(* Logix 5000 project; controller SX_V040001_C001 vendor 1 type 14 code 77 rev 16.23; software revision 16.04; part 10 of 35 *)
(* tags used below, declared in another part *)
   ALL_KINDS : INT[90];
   CMD : INT[36];
   command_value : INT;
   DATAOP : INT[10];
   DRIVE : INT[32];
   DRIVE_INTERVAL : INT[8];
   EMPTYING : INT[18];
   G_DInput : DINT[3];
   G_DOutput : DINT[3];
   loading : INT[19];
   louvre : INT[11];
   METERING : INT[44];
   METERING_PULSE : DINT[14];
   NOTDOS : INT[6];
   PARAMETER : INT[501];
   RECIPE_GENERAL : INT[405];
   RM_CMD : INT[9];
   T_CURRENT_EM_METER : TIMER;
   T_DELTA_EM_METER : TIMER;
   T_RPM_EM_METER : TIMER;
   T_TEMP_EM_METER : TIMER;
   TEMP : INT[14];
(* MainProgram, continued *)

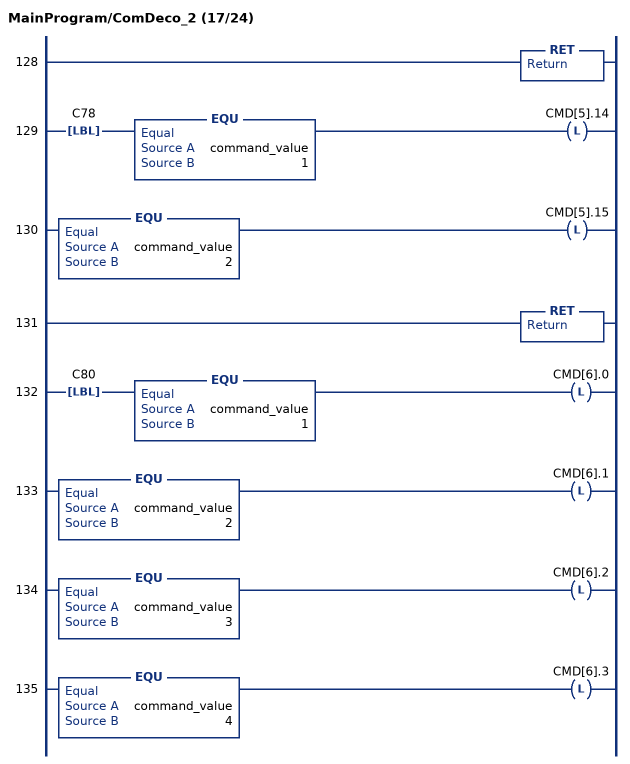
   [picture p205: MainProgram/ComDeco_2 rungs 128-135]
   128: RET();
   129: LBL(C78)EQU(command_value,1)OTL(CMD[5].14);
   130: EQU(command_value,2)OTL(CMD[5].15);
   131: RET();
   132: LBL(C80)EQU(command_value,1)OTL(CMD[6].0);
   133: EQU(command_value,2)OTL(CMD[6].1);
   134: EQU(command_value,3)OTL(CMD[6].2);
   135: EQU(command_value,4)OTL(CMD[6].3);
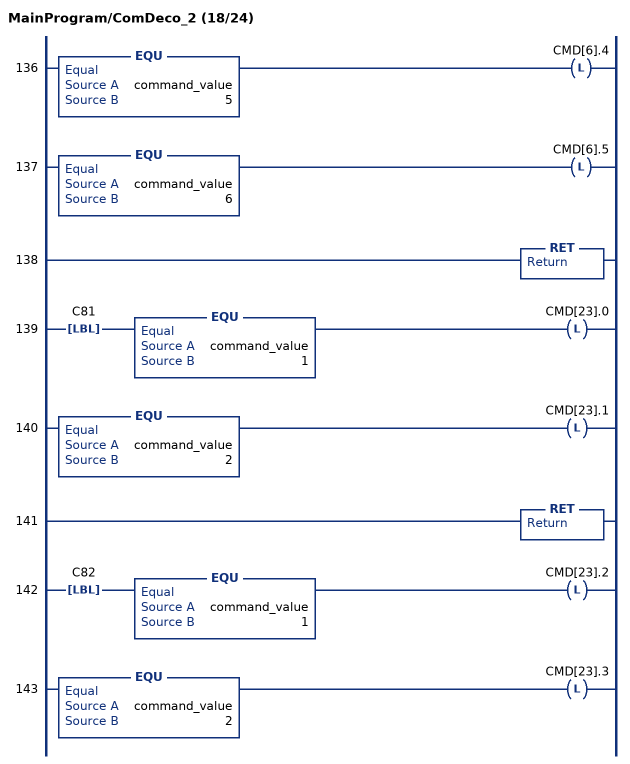
   136: EQU(command_value,5)OTL(CMD[6].4);
   137: EQU(command_value,6)OTL(CMD[6].5);
   138: RET();
   139: LBL(C81)EQU(command_value,1)OTL(CMD[23].0);
   140: EQU(command_value,2)OTL(CMD[23].1);
   141: RET();
   142: LBL(C82)EQU(command_value,1)OTL(CMD[23].2);
   143: EQU(command_value,2)OTL(CMD[23].3);
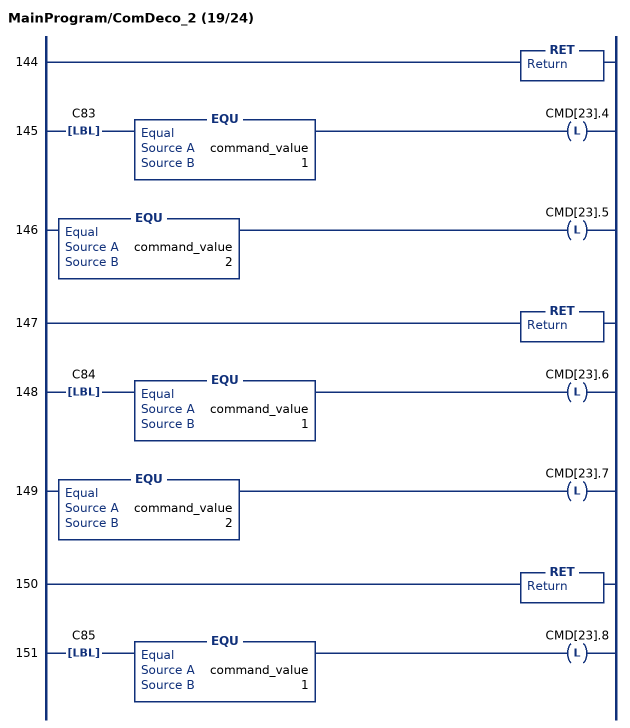
   144: RET();
   145: LBL(C83)EQU(command_value,1)OTL(CMD[23].4);
   146: EQU(command_value,2)OTL(CMD[23].5);
   147: RET();
   148: LBL(C84)EQU(command_value,1)OTL(CMD[23].6);
   149: EQU(command_value,2)OTL(CMD[23].7);
   150: RET();
   151: LBL(C85)EQU(command_value,1)OTL(CMD[23].8);
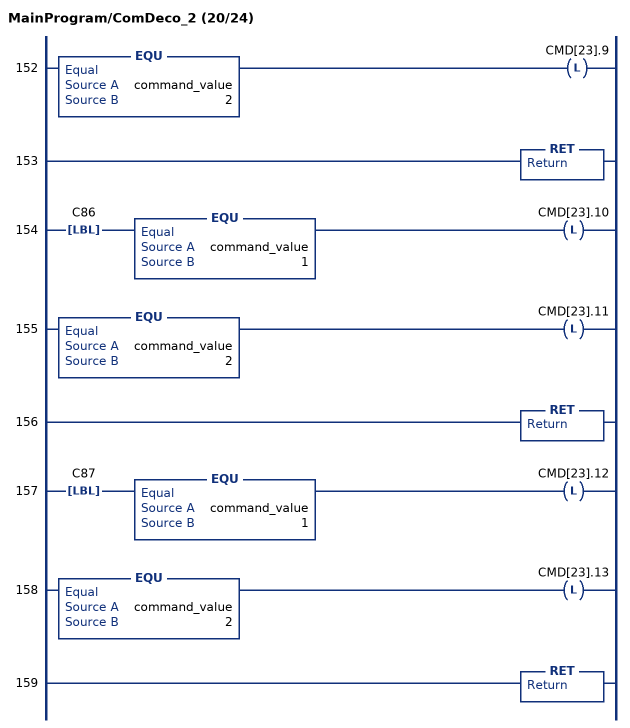
   152: EQU(command_value,2)OTL(CMD[23].9);
   153: RET();
   154: LBL(C86)EQU(command_value,1)OTL(CMD[23].10);
   155: EQU(command_value,2)OTL(CMD[23].11);
   156: RET();
   157: LBL(C87)EQU(command_value,1)OTL(CMD[23].12);
   158: EQU(command_value,2)OTL(CMD[23].13);
   159: RET();
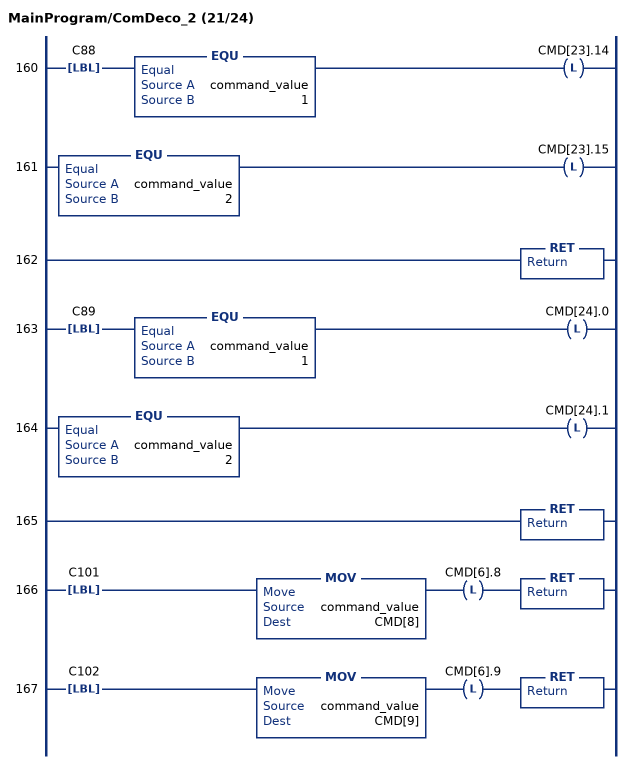
   160: LBL(C88)EQU(command_value,1)OTL(CMD[23].14);
   161: EQU(command_value,2)OTL(CMD[23].15);
   162: RET();
   163: LBL(C89)EQU(command_value,1)OTL(CMD[24].0);
   164: EQU(command_value,2)OTL(CMD[24].1);
   165: RET();
   166: LBL(C101)MOV(command_value,CMD[8])OTL(CMD[6].8)RET();
   167: LBL(C102)MOV(command_value,CMD[9])OTL(CMD[6].9)RET();
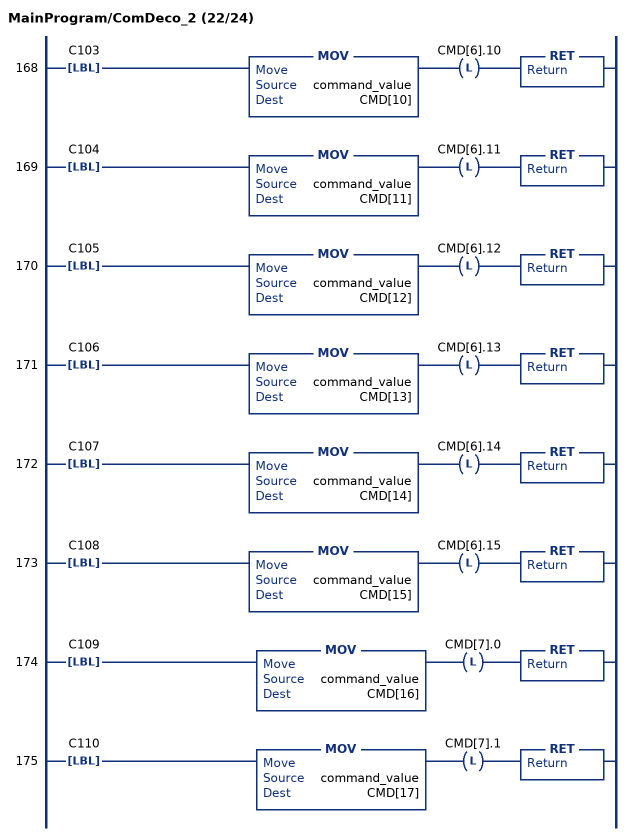
   168: LBL(C103)MOV(command_value,CMD[10])OTL(CMD[6].10)RET();
   169: LBL(C104)MOV(command_value,CMD[11])OTL(CMD[6].11)RET();
   170: LBL(C105)MOV(command_value,CMD[12])OTL(CMD[6].12)RET();
   171: LBL(C106)MOV(command_value,CMD[13])OTL(CMD[6].13)RET();
   172: LBL(C107)MOV(command_value,CMD[14])OTL(CMD[6].14)RET();
   173: LBL(C108)MOV(command_value,CMD[15])OTL(CMD[6].15)RET();
   174: LBL(C109)MOV(command_value,CMD[16])OTL(CMD[7].0)RET();
   175: LBL(C110)MOV(command_value,CMD[17])OTL(CMD[7].1)RET();
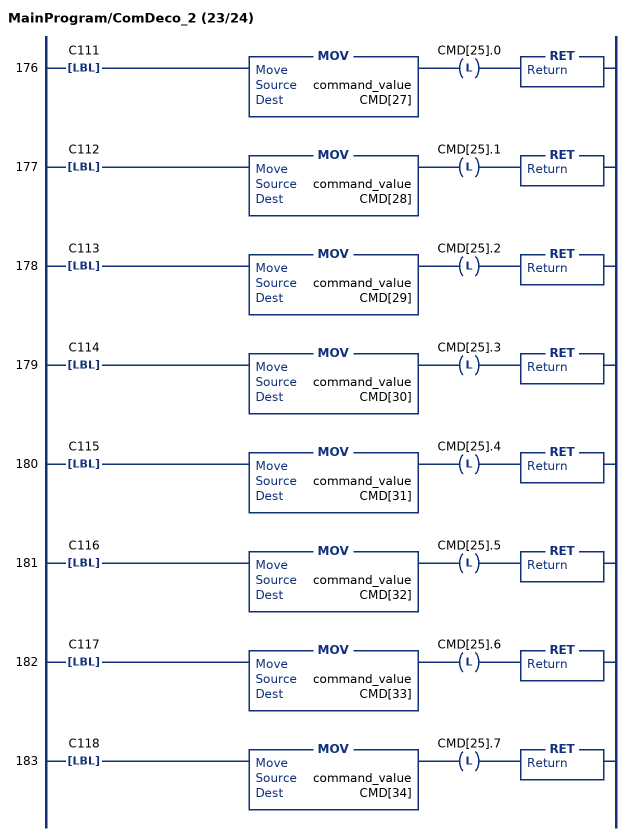
   176: LBL(C111)MOV(command_value,CMD[27])OTL(CMD[25].0)RET();
   177: LBL(C112)MOV(command_value,CMD[28])OTL(CMD[25].1)RET();
   178: LBL(C113)MOV(command_value,CMD[29])OTL(CMD[25].2)RET();
   179: LBL(C114)MOV(command_value,CMD[30])OTL(CMD[25].3)RET();
   180: LBL(C115)MOV(command_value,CMD[31])OTL(CMD[25].4)RET();
   181: LBL(C116)MOV(command_value,CMD[32])OTL(CMD[25].5)RET();
   182: LBL(C117)MOV(command_value,CMD[33])OTL(CMD[25].6)RET();
   183: LBL(C118)MOV(command_value,CMD[34])OTL(CMD[25].7)RET();
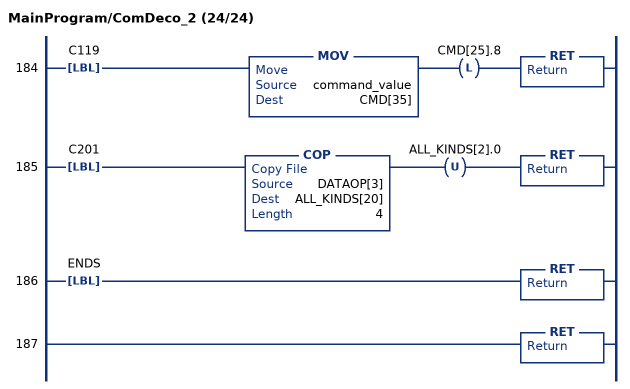
   184: LBL(C119)MOV(command_value,CMD[35])OTL(CMD[25].8)RET();
   185: LBL(C201)COP(DATAOP[3],ALL_KINDS[20],4)OTU(ALL_KINDS[2].0)RET();
   186: LBL(ENDS)RET();
   187: RET();
END_ROUTINE

ROUTINE DeleteData   (* ladder *)
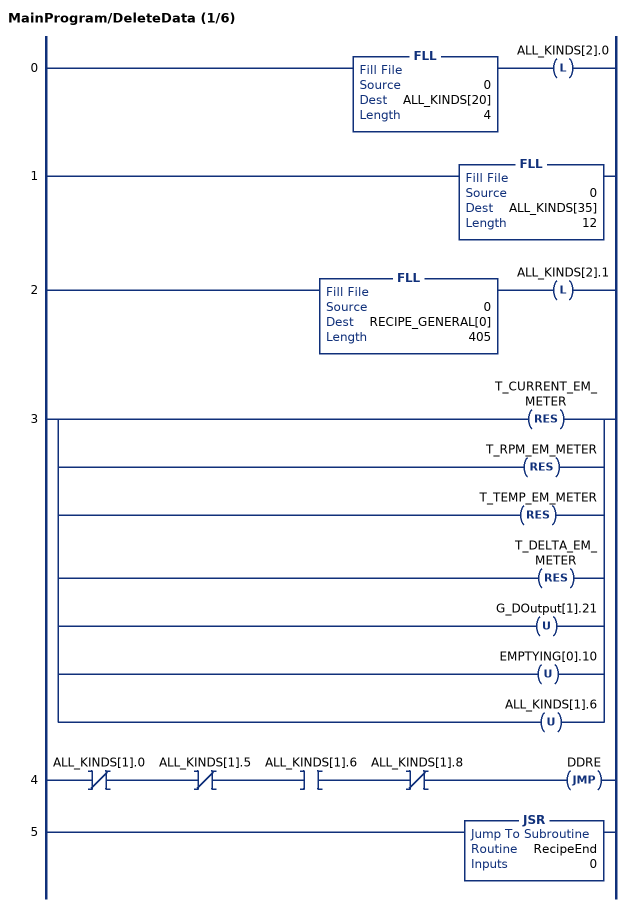
   0: FLL(0,ALL_KINDS[20],4)OTL(ALL_KINDS[2].0);
   1: FLL(0,ALL_KINDS[35],12);
   2: FLL(0,RECIPE_GENERAL[0],405)OTL(ALL_KINDS[2].1);
   3: [RES(T_CURRENT_EM_METER) ,RES(T_RPM_EM_METER) ,RES(T_TEMP_EM_METER) ,RES(T_DELTA_EM_METER) ,OTU(G_DOutput[1].21) ,OTU(EMPTYING[0].10) ,OTU(ALL_KINDS[1].6) ];
   4: XIO(ALL_KINDS[1].0)XIO(ALL_KINDS[1].5)XIC(ALL_KINDS[1].6)XIO(ALL_KINDS[1].8)JMP(DDRE);
   5: JSR(RecipeEnd,0);
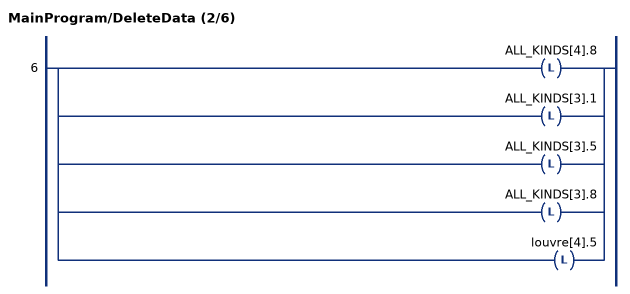
   6: [OTL(ALL_KINDS[4].8) ,OTL(ALL_KINDS[3].1) ,OTL(ALL_KINDS[3].5) ,OTL(ALL_KINDS[3].8) ,OTL(louvre[4].5) ];
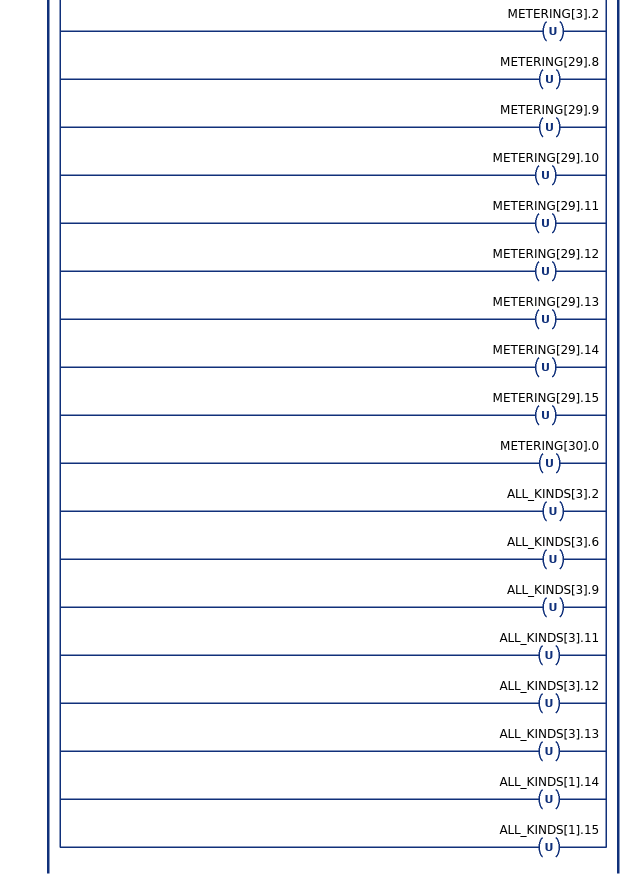
   7: [OTU(ALL_KINDS[4].9) ,OTU(ALL_KINDS[1].3) ,OTU(ALL_KINDS[3].5) ,OTU(ALL_KINDS[1].5) ,OTU(ALL_KINDS[1].7) ,OTU(ALL_KINDS[1].8) ,OTU(ALL_KINDS[1].9) ,OTU(RM_CMD[3].1) ,OTU(ALL_KINDS[1].11) ,OTU(ALL_KINDS[1].12) ,OTU(ALL_KINDS[1].13) ,OTU(ALL_KINDS[2].2) ,OTU(ALL_KINDS[2].4) ,OTU(METERING[2].5) ,OTU(METERING[2].6) ,OTU(EMPTYING[1].9) ,OTU(DRIVE[2].4) ,OTU(DRIVE_INTERVAL[1].0) ,OTU(EMPTYING[0].15) ,OTU(EMPTYING[1].15) ,OTU(TEMP[1].2) ,OTU(loading[1].1) ,OTU(NOTDOS[1].0) ,OTU(NOTDOS[1].7) ,OTU(NOTDOS[1].9) ,OTU(NOTDOS[1].1) ,OTU(NOTDOS[1].8) ,OTU(NOTDOS[1].10) ,OTU(NOTDOS[1].2) ,OTU(NOTDOS[1].3) ,OTU(NOTDOS[1].4) ,OTU(NOTDOS[1].5) ,OTU(NOTDOS[1].6) ,OTU(METERING[1].0) ,OTU(METERING[1].1) ,OTU(METERING[1].2) ,OTU(METERING[1].3) ,OTU(METERING[1].4) ,OTU(METERING[27].0) ,OTU(METERING[27].1) ,OTU(METERING[27].2) ,OTU(METERING[27].3) ,OTU(METERING[27].4) ,OTU(METERING[27].5) ,OTU(METERING[27].6) ,OTU(METERING[27].7) ,OTU(METERING[27].8) ,OTU(METERING[1].10) ,OTU(METERING[1].11) ,OTU(METERING[1].12) ,OTU(METERING[1].13) ,OTU(METERING[1].14) ,OTU(METERING[28].4) ,OTU(METERING[28].5) ,OTU(METERING[28].6) ,OTU(METERING[28].7) ,OTU(METERING[28].8) ,OTU(METERING[28].9) ,OTU(METERING[28].10) ,OTU(METERING[28].11) ,OTU(METERING[28].12) ,OTU(METERING[2].14) ,OTU(METERING[2].15) ,OTU(METERING[3].0) ,OTU(METERING[3].1) ,OTU(METERING[3].2) ,OTU(METERING[29].8) ,OTU(METERING[29].9) ,OTU(METERING[29].10) ,OTU(METERING[29].11) ,OTU(METERING[29].12) ,OTU(METERING[29].13) ,OTU(METERING[29].14) ,OTU(METERING[29].15) ,OTU(METERING[30].0) ,OTU(ALL_KINDS[3].2) ,OTU(ALL_KINDS[3].6) ,OTU(ALL_KINDS[3].9) ,OTU(ALL_KINDS[3].11) ,OTU(ALL_KINDS[3].12) ,OTU(ALL_KINDS[3].13) ,OTU(ALL_KINDS[1].14) ,OTU(ALL_KINDS[1].15) ];
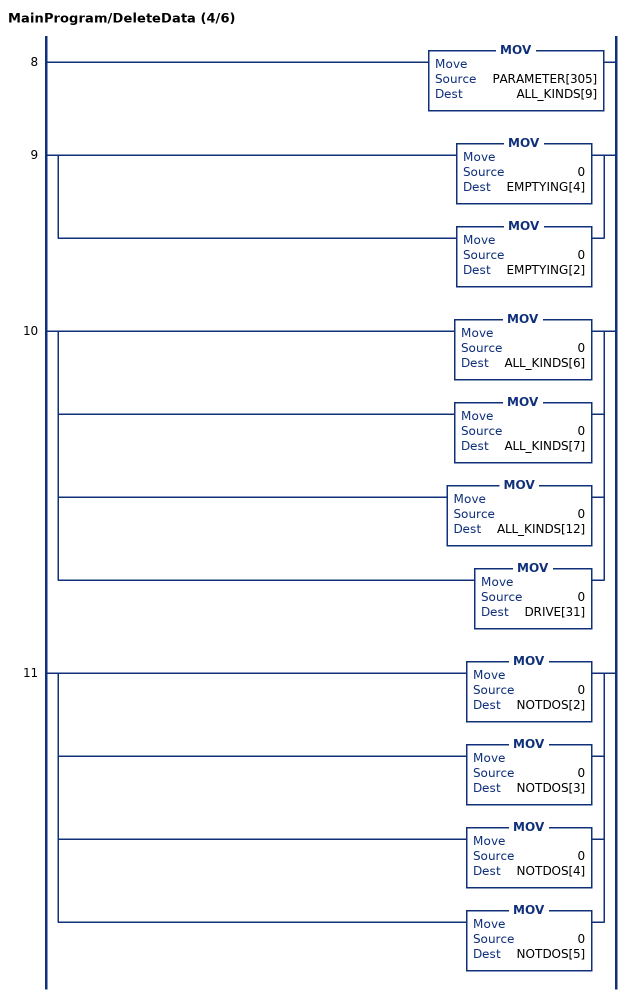
   8: MOV(PARAMETER[305],ALL_KINDS[9]);
   9: [MOV(0,EMPTYING[4]) ,MOV(0,EMPTYING[2]) ];
   10: [MOV(0,ALL_KINDS[6]) ,MOV(0,ALL_KINDS[7]) ,MOV(0,ALL_KINDS[12]) ,MOV(0,DRIVE[31]) ];
   11: [MOV(0,NOTDOS[2]) ,MOV(0,NOTDOS[3]) ,MOV(0,NOTDOS[4]) ,MOV(0,NOTDOS[5]) ];
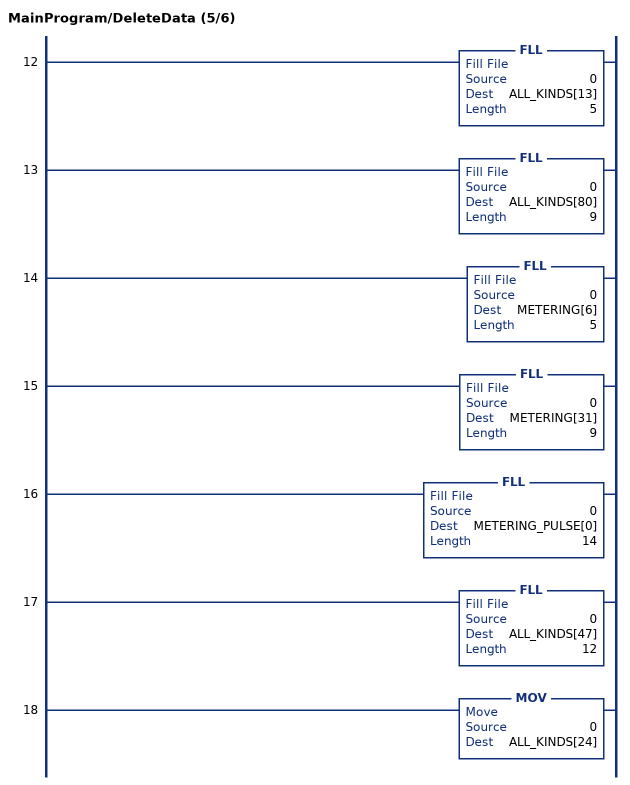
   12: FLL(0,ALL_KINDS[13],5);
   13: FLL(0,ALL_KINDS[80],9);
   14: FLL(0,METERING[6],5);
   15: FLL(0,METERING[31],9);
   16: FLL(0,METERING_PULSE[0],14);
   17: FLL(0,ALL_KINDS[47],12);
   18: MOV(0,ALL_KINDS[24]);
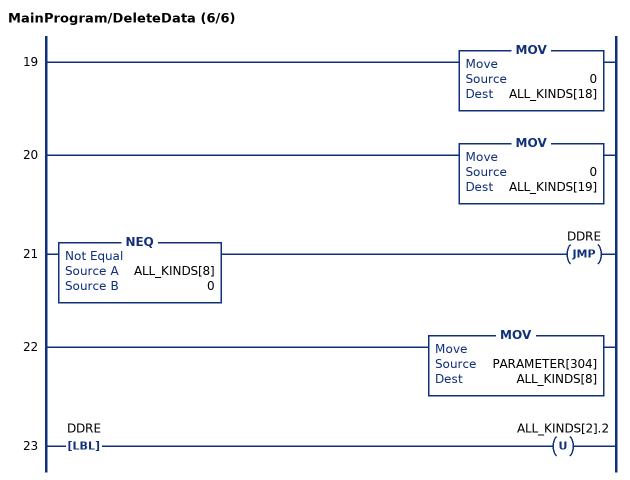
   19: MOV(0,ALL_KINDS[18]);
   20: MOV(0,ALL_KINDS[19]);
   21: NEQ(ALL_KINDS[8],0)JMP(DDRE);
   22: MOV(PARAMETER[304],ALL_KINDS[8]);
   23: LBL(DDRE)OTU(ALL_KINDS[2].2);
END_ROUTINE

ROUTINE DomELK   (* ladder *)
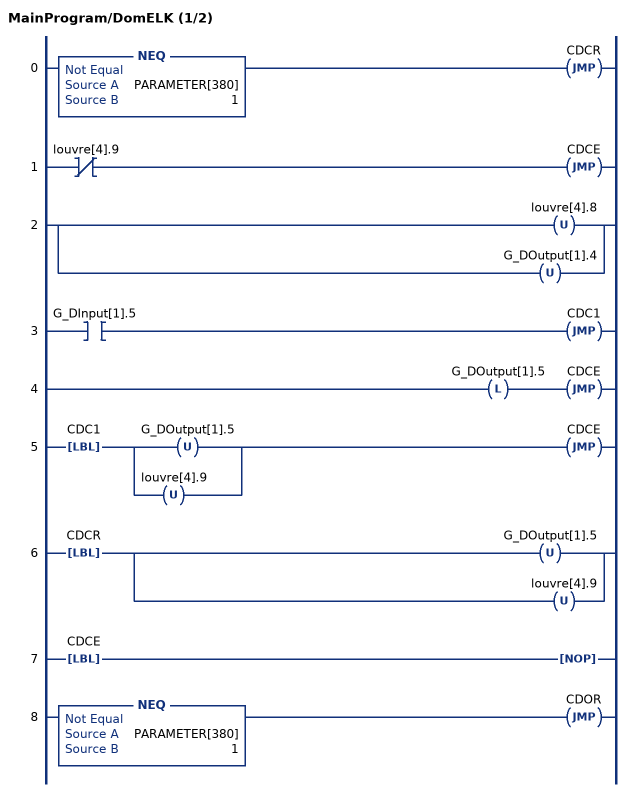
   0: NEQ(PARAMETER[380],1)JMP(CDCR);
   1: XIO(louvre[4].9)JMP(CDCE);
   2: [OTU(louvre[4].8) ,OTU(G_DOutput[1].4) ];
   3: XIC(G_DInput[1].5)JMP(CDC1);
   4: OTL(G_DOutput[1].5)JMP(CDCE);
   5: LBL(CDC1)[OTU(G_DOutput[1].5) ,OTU(louvre[4].9) ]JMP(CDCE);
   6: LBL(CDCR)[OTU(G_DOutput[1].5) ,OTU(louvre[4].9) ];
   7: LBL(CDCE)NOP();
   8: NEQ(PARAMETER[380],1)JMP(CDOR);
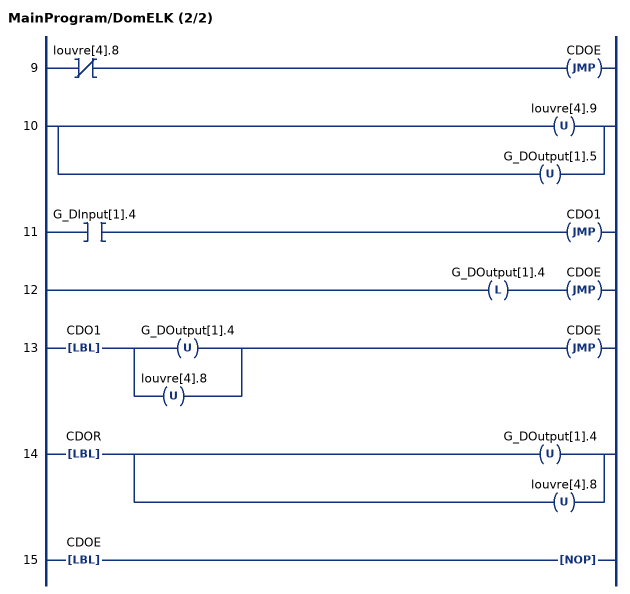
   9: XIO(louvre[4].8)JMP(CDOE);
   10: [OTU(louvre[4].9) ,OTU(G_DOutput[1].5) ];
   11: XIC(G_DInput[1].4)JMP(CDO1);
   12: OTL(G_DOutput[1].4)JMP(CDOE);
   13: LBL(CDO1)[OTU(G_DOutput[1].4) ,OTU(louvre[4].8) ]JMP(CDOE);
   14: LBL(CDOR)[OTU(G_DOutput[1].4) ,OTU(louvre[4].8) ];
   15: LBL(CDOE)NOP();
END_ROUTINE

ROUTINE EmergencyMetering   (* ladder *)
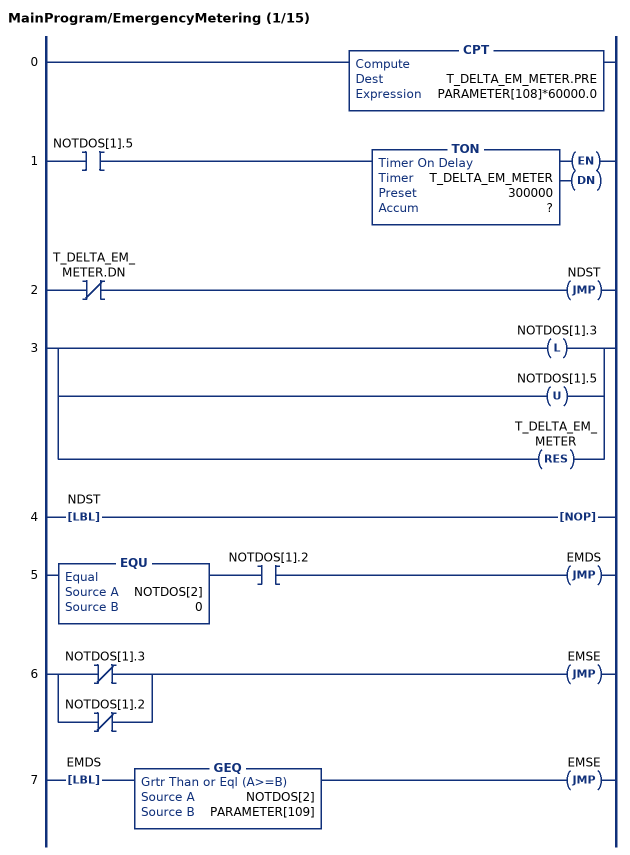
   0: CPT(T_DELTA_EM_METER.PRE,PARAMETER[108]*60000.0);
   1: XIC(NOTDOS[1].5)TON(T_DELTA_EM_METER,?,?);
   2: XIO(T_DELTA_EM_METER.DN)JMP(NDST);
   3: [OTL(NOTDOS[1].3) ,OTU(NOTDOS[1].5) ,RES(T_DELTA_EM_METER) ];
   4: LBL(NDST)NOP();
   5: EQU(NOTDOS[2],0)XIC(NOTDOS[1].2)JMP(EMDS);
   6: [XIO(NOTDOS[1].3) ,XIO(NOTDOS[1].2) ]JMP(EMSE);
   7: LBL(EMDS)GEQ(NOTDOS[2],PARAMETER[109])JMP(EMSE);
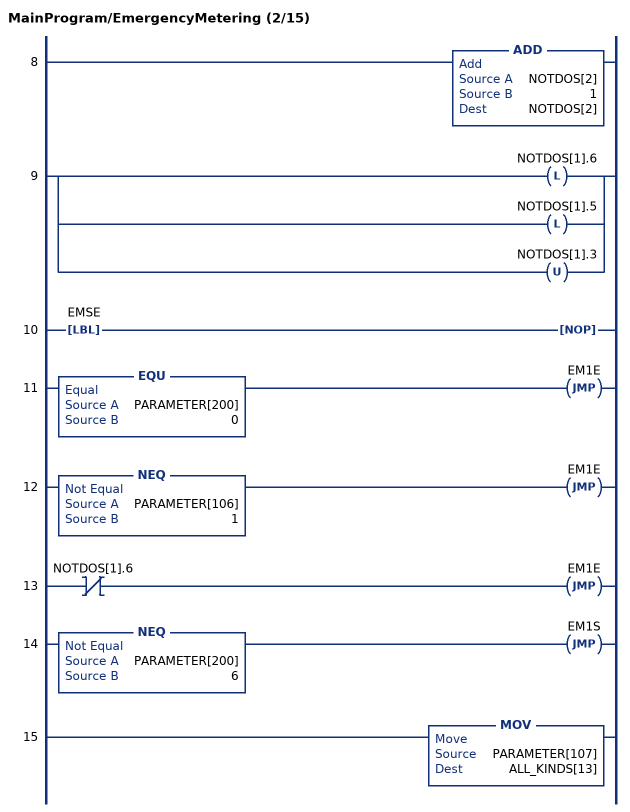
   8: ADD(NOTDOS[2],1,NOTDOS[2]);
   9: [OTL(NOTDOS[1].6) ,OTL(NOTDOS[1].5) ,OTU(NOTDOS[1].3) ];
   10: LBL(EMSE)NOP();
   11: EQU(PARAMETER[200],0)JMP(EM1E);
   12: NEQ(PARAMETER[106],1)JMP(EM1E);
   13: XIO(NOTDOS[1].6)JMP(EM1E);
   14: NEQ(PARAMETER[200],6)JMP(EM1S);
   15: MOV(PARAMETER[107],ALL_KINDS[13]);
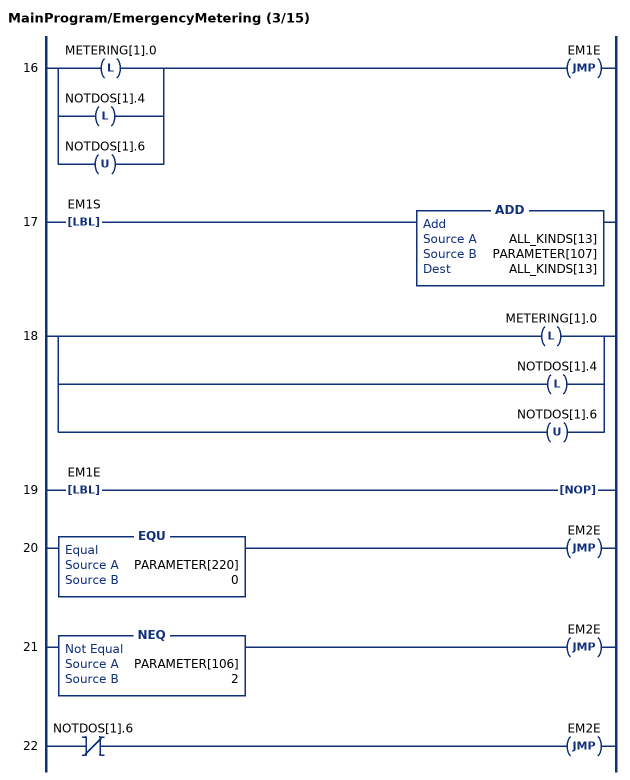
   16: [OTL(METERING[1].0) ,OTL(NOTDOS[1].4) ,OTU(NOTDOS[1].6) ]JMP(EM1E);
   17: LBL(EM1S)ADD(ALL_KINDS[13],PARAMETER[107],ALL_KINDS[13]);
   18: [OTL(METERING[1].0) ,OTL(NOTDOS[1].4) ,OTU(NOTDOS[1].6) ];
   19: LBL(EM1E)NOP();
   20: EQU(PARAMETER[220],0)JMP(EM2E);
   21: NEQ(PARAMETER[106],2)JMP(EM2E);
   22: XIO(NOTDOS[1].6)JMP(EM2E);
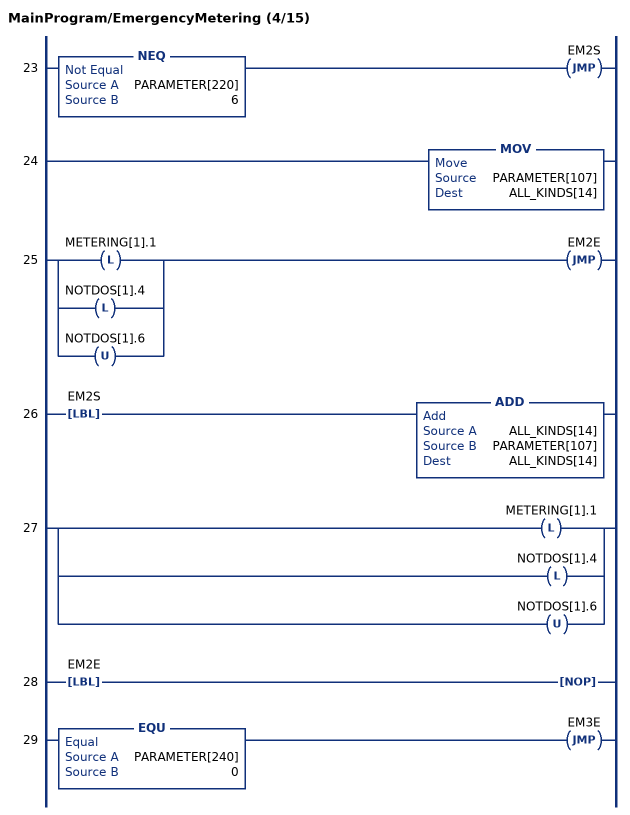
   23: NEQ(PARAMETER[220],6)JMP(EM2S);
   24: MOV(PARAMETER[107],ALL_KINDS[14]);
   25: [OTL(METERING[1].1) ,OTL(NOTDOS[1].4) ,OTU(NOTDOS[1].6) ]JMP(EM2E);
   26: LBL(EM2S)ADD(ALL_KINDS[14],PARAMETER[107],ALL_KINDS[14]);
   27: [OTL(METERING[1].1) ,OTL(NOTDOS[1].4) ,OTU(NOTDOS[1].6) ];
   28: LBL(EM2E)NOP();
   29: EQU(PARAMETER[240],0)JMP(EM3E);
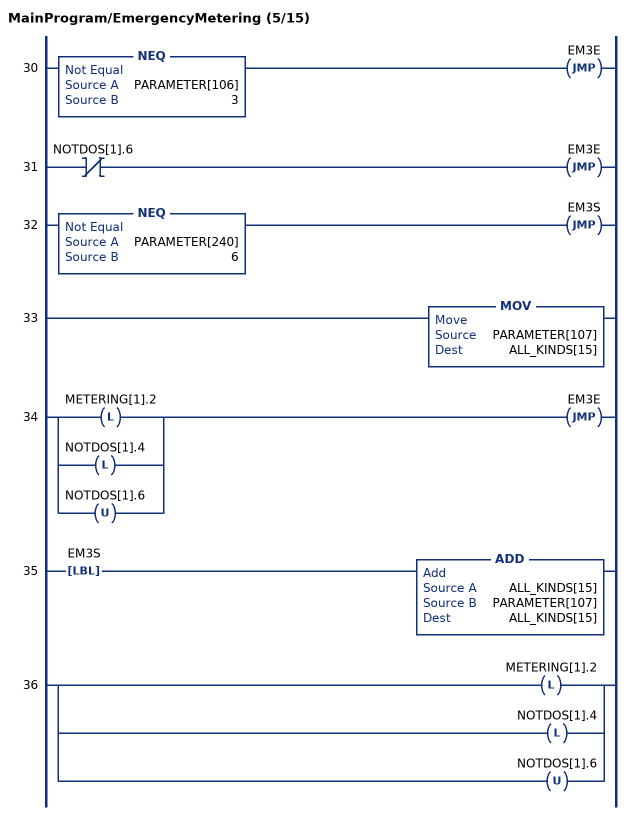
   30: NEQ(PARAMETER[106],3)JMP(EM3E);
   31: XIO(NOTDOS[1].6)JMP(EM3E);
   32: NEQ(PARAMETER[240],6)JMP(EM3S);
   33: MOV(PARAMETER[107],ALL_KINDS[15]);
   34: [OTL(METERING[1].2) ,OTL(NOTDOS[1].4) ,OTU(NOTDOS[1].6) ]JMP(EM3E);
   35: LBL(EM3S)ADD(ALL_KINDS[15],PARAMETER[107],ALL_KINDS[15]);
   36: [OTL(METERING[1].2) ,OTL(NOTDOS[1].4) ,OTU(NOTDOS[1].6) ];
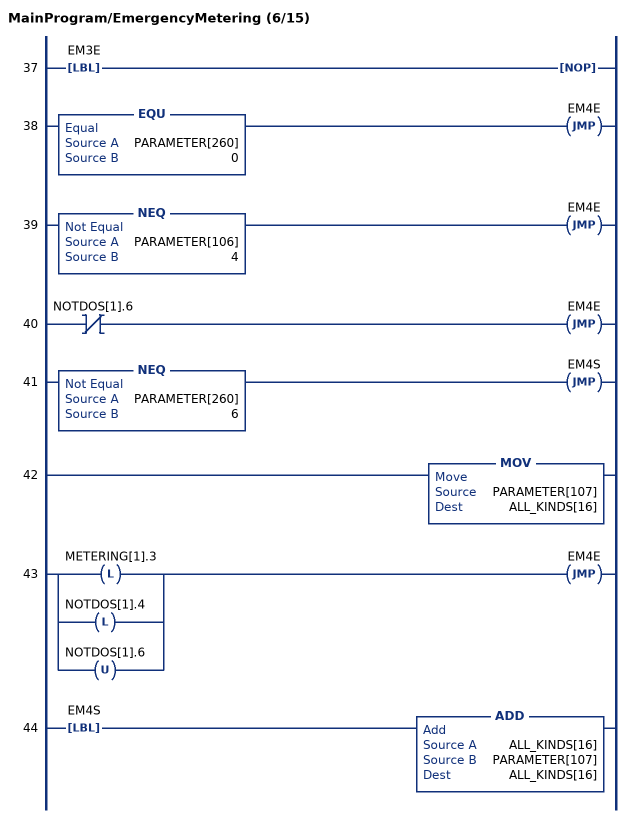
   37: LBL(EM3E)NOP();
   38: EQU(PARAMETER[260],0)JMP(EM4E);
   39: NEQ(PARAMETER[106],4)JMP(EM4E);
   40: XIO(NOTDOS[1].6)JMP(EM4E);
   41: NEQ(PARAMETER[260],6)JMP(EM4S);
   42: MOV(PARAMETER[107],ALL_KINDS[16]);
   43: [OTL(METERING[1].3) ,OTL(NOTDOS[1].4) ,OTU(NOTDOS[1].6) ]JMP(EM4E);
   44: LBL(EM4S)ADD(ALL_KINDS[16],PARAMETER[107],ALL_KINDS[16]);
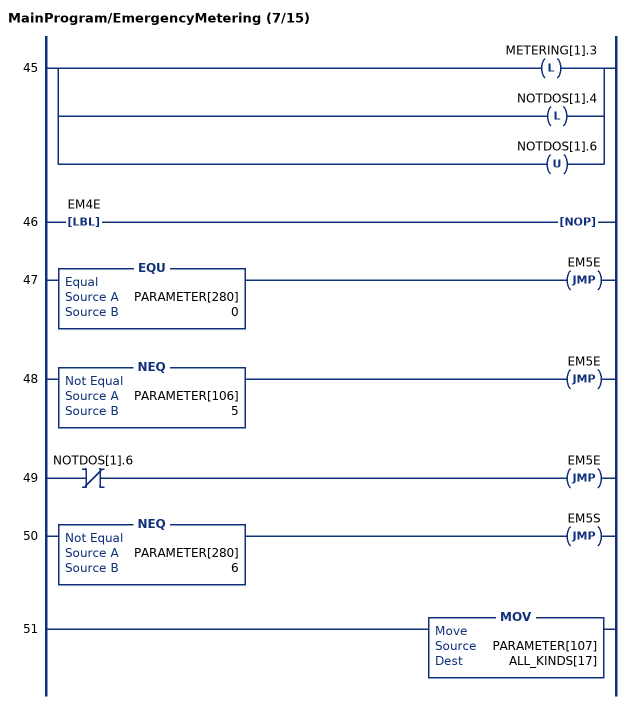
   45: [OTL(METERING[1].3) ,OTL(NOTDOS[1].4) ,OTU(NOTDOS[1].6) ];
   46: LBL(EM4E)NOP();
   47: EQU(PARAMETER[280],0)JMP(EM5E);
   48: NEQ(PARAMETER[106],5)JMP(EM5E);
   49: XIO(NOTDOS[1].6)JMP(EM5E);
   50: NEQ(PARAMETER[280],6)JMP(EM5S);
   51: MOV(PARAMETER[107],ALL_KINDS[17]);
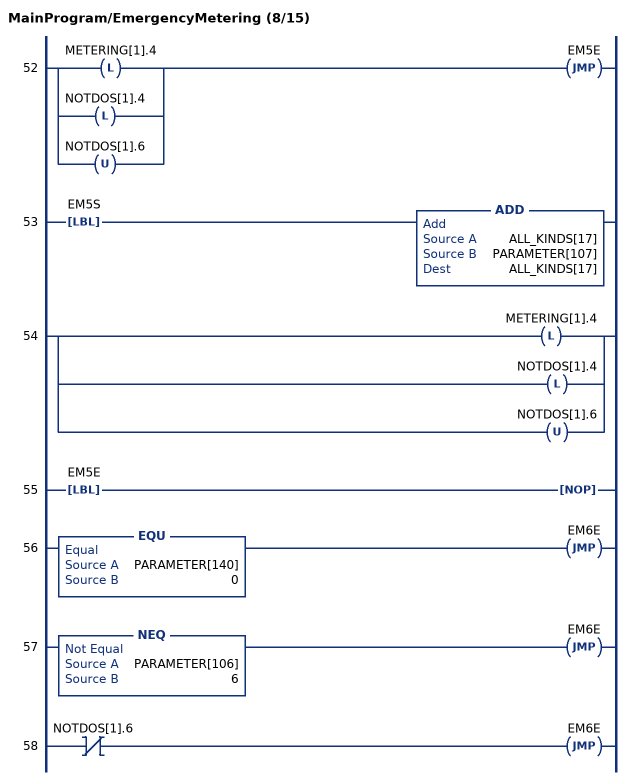
   52: [OTL(METERING[1].4) ,OTL(NOTDOS[1].4) ,OTU(NOTDOS[1].6) ]JMP(EM5E);
   53: LBL(EM5S)ADD(ALL_KINDS[17],PARAMETER[107],ALL_KINDS[17]);
   54: [OTL(METERING[1].4) ,OTL(NOTDOS[1].4) ,OTU(NOTDOS[1].6) ];
   55: LBL(EM5E)NOP();
   56: EQU(PARAMETER[140],0)JMP(EM6E);
   57: NEQ(PARAMETER[106],6)JMP(EM6E);
   58: XIO(NOTDOS[1].6)JMP(EM6E);
